PROGRAM MAIN
VAR
	
	{attribute 'OPC.UA.DA':='1'}
	Piezo001:		FB_PIEZO_EXAMPLE;	// Piezo #1
	{attribute 'OPC.UA.DA':='1'}
	Piezo002:		FB_PIEZO_EXAMPLE;	// Piezo #2
	
	{attribute 'OPC.UA.DA':='1'}
	SIM_Piezo001:	FB_SIM_PIEZO;		// Simulator for Piezo #1 (if simulated)
	{attribute 'OPC.UA.DA':='1'}
	SIM_Piezo002:	FB_SIM_PIEZO;		// Simulator for Piezo #2 (always simulated)

END_VAR

Piezo001(in_sName:='Piezo001', in_nNumAxes:=3);

Piezo002(in_sName:='Piezo002', in_nNumAxes:=3);

SIM_Piezo001();
SIM_Piezo002();

END_PROGRAM

(* stored: Version 1.1.0.1, ProductVersion 3.1.4024.3
   POU MAIN: Id {4e85b569-c316-4f2d-ac6b-3e20253d8a12}, SpecialFunc None *)
